(* CODESYS project PresentBagSequence.xml

Project tree, tasks and I/O mapping:
  function block PresentBagSequence [SFC]
*)

// PresentBagSequence
FUNCTION_BLOCK PresentBagSequence
VAR_INPUT
	SFCInit: BOOL;
	Trigger: BOOL;
	KickerRaised: BOOL;
	KickerLowered: BOOL;
END_VAR
VAR_OUTPUT
	RaiseKicker: BOOL;
	LowerKicker: BOOL;
END_VAR
VAR
END_VAR

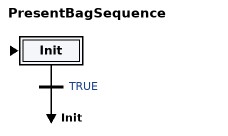
INITIAL_STEP Init:
END_STEP
TRANSITION FROM Init TO Init
    := TRUE;
END_TRANSITION

END_FUNCTION_BLOCK
